FUNCTION_BLOCK EcMasterProtocolError IMPLEMENTS IEcTask
VAR_INPUT
END_VAR
VAR_OUTPUT
END_VAR
VAR
	iState : INT;
	masterProtocolErr : Tc2_EtherCAT.FB_EcGetLastProtErrInfo;
	_execute: BOOL;
	_done: BOOL;
	_busy: BOOL;
	_error: BOOL;
	_netId: AMSNETID;
END_VAR

CASE iState OF
	0:
		IF _execute THEN
			_done := FALSE;
			_busy := TRUE;
			_error := FALSE;
			masterProtocolErr.bExecute := TRUE;
			IF masterProtocolErr.bBusy THEN
				iState := 10;
				_execute := false;
			END_IF
		END_IF
	10:
		IF NOT masterProtocolErr.bBusy THEN
			IF NOT masterProtocolErr.bError THEN
				_done := TRUE;
			ELSE
				_error := TRUE;
			END_IF
			_busy := FALSE;
			masterProtocolErr.bExecute := FALSE;
			iState := 0;
		END_IF
END_CASE

masterProtocolErr(sNetId := Tc2_System.F_CreateAmsNetId(nIds := NetId));

{warning 'add method implementation '}
METHOD Abort : BOOL
masterProtocolErr.bExecute := FALSE;
_busy := FALSE;
_execute := FALSE;
Abort := TRUE;
iState := 0;
END_METHOD

{warning 'add property implementation'}
PROPERTY Busy : BOOL
GET
Busy := _busy;
END_GET
END_PROPERTY

PROPERTY DeviceAddr : uint
GET
DeviceAddr := masterProtocolErr.nSlaveAddr;
END_GET
SET
masterProtocolErr.nSlaveAddr := DeviceAddr;
END_SET
END_PROPERTY

{warning 'add property implementation'}
PROPERTY Done : BOOL
GET
Done := _done;
END_GET
END_PROPERTY

{warning 'add property implementation'}
PROPERTY Error : BOOL
GET
Error := _error;
END_GET
END_PROPERTY

{warning 'add method implementation '}
METHOD Execute : BOOL
IF NOT masterProtocolErr.bBusy THEN
	Execute := _execute := TRUE;
END_IF
END_METHOD

PROPERTY LastProtocolError : ST_EcLastProtErrInfo
GET
LastProtocolError := masterProtocolErr.info;
END_GET
END_PROPERTY

{warning 'add property implementation'}
PROPERTY NetID : amsnetid
GET
NetID := _netId;
END_GET
SET
_netId := NetID;
END_SET
END_PROPERTY

PROPERTY ProtocolType : E_EcMbxProtType
GET
ProtocolType := masterProtocolErr.eProtocol;
END_GET
SET
masterProtocolErr.eProtocol := ProtocolType;
END_SET
END_PROPERTY

END_FUNCTION_BLOCK

(* stored: Version 1.1.0.1, ProductVersion 3.1.4024.11
   POU EcMasterProtocolError: Id {e8b7c2a1-d525-4c66-9331-a9766493620c}, SpecialFunc None
   Method Abort: Id {94be40df-127e-4d97-8546-306373d103ba}
   Property Busy: Id {de9102ad-58f8-45ba-9c6c-ccbb276256c1}
   Get Get: Id {50bf087d-3cfc-433f-a6a6-02db096ade9c}
   Property DeviceAddr: Id {b290b5b3-83d0-4711-aa82-add5e8ad6dcb}
   Get Get: Id {bb8f11b5-b665-40e5-9331-a929c67f83b3}
   Set Set: Id {dad4e2d0-6cc3-4d69-8745-1834f457906d}
   Property Done: Id {30df4c4a-2ccc-40e0-a04f-d2b3073d604d}
   Get Get: Id {7dbcfda0-c022-4b5a-8b5f-181a78e62b3f}
   Property Error: Id {55c53937-8cf8-43f5-8695-c18ab1685ef2}
   Get Get: Id {35fed673-4440-4a9f-9423-b5ea129b6935}
   Method Execute: Id {8f873a0b-714d-4078-b4dd-ebcc940ba281}
   Property LastProtocolError: Id {a1990021-535c-4c44-95d7-f13fe0829f4d}
   Get Get: Id {7903afc8-23ac-42e9-8458-66f5e5597de8}
   Property NetID: Id {19b727cb-3117-4097-98f5-7787868cd1b5}
   Get Get: Id {8d064c2e-41ce-425f-b4c9-e9627fa289fb}
   Set Set: Id {abe475f4-c4e3-411e-abd3-f84ddeb31b8f}
   Property ProtocolType: Id {75085b6f-8630-466e-b399-6a68a44cee29}
   Get Get: Id {62db3fec-8dea-4156-a618-721d2e01db7b}
   Set Set: Id {ba07eb36-7b1a-461a-b728-ed447595209b} *)
